(* CODESYS project SZ10-12 PROJ.project

Project tree, tasks and I/O mapping:
  Device : CPX-CEC-S1-V3, Festo AG & Co. KG, order no. 3472425, version 3.5.7.37
      unmapped channels: Rotary switch
    application Application
      libraries: Standard, * (System)
      task MainTask (cyclic, interval t#20ms, priority 20) calls PLC_PRG
      program PLC_PRG [SFC]: Step0_active, Step7_active, Step1_active, Step2_active, Step3_active, Step4_active, Step6_active, Step5_active, Step8_active, Init_active, Step9_active, Step10_active, Step11_active, Step12_active, Step14_active, Step15_active, Step16_active, Step17_active, Step18_active, Step19_active, Step20_active, Step21_active, Step30_active, Step31_active, Step32_active, Step33_active, Step36_active
      global variables GVL
    PLC_Diagnosis : PLC-Diagnosis, Festo AG & Co. KG, version 3.5.4.1
    CPX_System : CPX_System, Festo AG & Co. KG, order no. 3472425, version 1.258
      CEC_S1_V3 : CEC-S1-V3, Festo AG & Co. KG, order no. 3472425, version 1.258
          settings:  = 0;  = 169055699865088;  = 1107404992;  = 16777215;  = 16885952;  = 13959210;  = 1f58c199;  = 5
      _8DI_8DO : 8DI/8DO, Festo AG & Co. KG, order no. 526257, version 1.258
          settings:  = 0;  = 1;  = 1;  = 1;  = 1;  = 0;  = 1;  = 1;  = 0;  = 0;  = 0;  = 0;  = 0;  = 0;  = 0;  = 0;  = 0;  = 0;  = 0;  = 0;  = 0;  = 0;  = 0;  = 0;  = 0;  = 0;  = 0;  = 0;  = 0;  = 0;  = 0;  = 0;  = 0;  = 0;  = 0;  = 0;  = 0;  = 0;  = 0;  = 0;
             = 0;  = 0;  = 0;  = 0;  = 0;  = 0;  = 0;  = 0;  = 0;  = 0;  = 0;  = 0;  = 0;  = 0;  = 0;  = 0;  = 0;  = 0;  = 0;  = 0;  = 0;  = 0;  = 0;  = 0;  = 0;  = 0;  = 0;  = 0;  = 0;  = 0;  = 0;  = 0;  = 0;  = 0;  = 0;  = 0;  = 0;  = 0;  = 0;  = 0;
             = 576751027668385792;  = 'PI%i.0.0.1=1';  = 'PI%i.0.1.1=1';  = 'PI%i.0.2.1=1';  = 'PI%i.1.0.1=1';  = 'PI%i.1.1.1=0';  = 'PI%i.1.4.2=1';  = 'PI%i.1.6.2=1';  = 'PI%i.6.0.1=0';  = 'PI%i.6.1.1=0';  = 'PI%i.6.2.1=0';  = 'PI%i.6.3.1=0';  = 'PI%i.6.4.1=0';  = 'PI%i.6.5.1=0';  = 'PI%i.6.6.1=0';  = 'PI%i.6.7.1=0';  = dd3e3128;  = 6
          unmapped channels: Input 0, Output 0
      _8DI_8DO_1 : 8DI/8DO, Festo AG & Co. KG, order no. 526257, version 1.258
          settings:  = 0;  = 1;  = 1;  = 1;  = 1;  = 0;  = 1;  = 1;  = 0;  = 0;  = 0;  = 0;  = 0;  = 0;  = 0;  = 0;  = 0;  = 0;  = 0;  = 0;  = 0;  = 0;  = 0;  = 0;  = 0;  = 0;  = 0;  = 0;  = 0;  = 0;  = 0;  = 0;  = 0;  = 0;  = 0;  = 0;  = 0;  = 0;  = 0;  = 0;
             = 0;  = 0;  = 0;  = 0;  = 0;  = 0;  = 0;  = 0;  = 0;  = 0;  = 0;  = 0;  = 0;  = 0;  = 0;  = 0;  = 0;  = 0;  = 0;  = 0;  = 0;  = 0;  = 0;  = 0;  = 0;  = 0;  = 0;  = 0;  = 0;  = 0;  = 0;  = 0;  = 0;  = 0;  = 0;  = 0;  = 0;  = 0;  = 0;  = 0;
             = 576751027668385792;  = 'PI%i.0.0.1=1';  = 'PI%i.0.1.1=1';  = 'PI%i.0.2.1=1';  = 'PI%i.1.0.1=1';  = 'PI%i.1.1.1=0';  = 'PI%i.1.4.2=1';  = 'PI%i.1.6.2=1';  = 'PI%i.6.0.1=0';  = 'PI%i.6.1.1=0';  = 'PI%i.6.2.1=0';  = 'PI%i.6.3.1=0';  = 'PI%i.6.4.1=0';  = 'PI%i.6.5.1=0';  = 'PI%i.6.6.1=0';  = 'PI%i.6.7.1=0';  = dd3e312f;  = 6
          unmapped channels: Input 0, Output 0
      _2AI : 2AI, Festo AG & Co. KG, order no. 526168, version 1.258
          settings:  = 0;  = 1;  = 1;  = 1;  = 1;  = 128;  = 128;  = 0;  = 0;  = 0;  = 0;  = 0;  = 0;  = 4095;  = 4095;  = 0;  = 0;  = 0;  = 0;  = 148618787711614976;  = 'PI%i.0.0.1=1';  = 'PI%i.0.7.1=1';  = 'PI%i.1.0.1=1';  = 'PI%i.3.0.2=1';  = 'PI%i.6.0.8=128';  = 'PI%i.7.0.8=128';  = 'PI%i.8.0.4=0';  = 'PI%i.8.4.4=0';  = 'PI%i.9.0.4=0';  = 'PI%i.9.4.4=0';  = 'PI%i.10.0.16=0';  = 'PI%i.12.0.16=0';  = 'PI%i.14.0.16=4095';  = 'PI%i.16.0.16=4095';  = dd3e2ea6;  = 15
          unmapped channels: Input 0, Input 1
      _2AO : 2AO, Festo AG & Co. KG, order no. 526170, version 1.258
          settings:  = 0;  = 1;  = 1;  = 1;  = 0;  = 1;  = 135;  = 135;  = 0;  = 0;  = 0;  = 0;  = 4095;  = 4095;  = 0;  = 0;  = 0;  = 0;  = 0;  = 0;  = 0;  = 0;  = 0;  = 0;  = 0;  = 0;  = 2267751186432;  = 'PI%i.0.1.1=1';  = 'PI%i.0.7.1=1';  = 'PI%i.1.1.1=1';  = 'PI%i.1.3.1=0';  = 'PI%i.3.4.2=1';  = 'PI%i.6.0.8=135';  = 'PI%i.7.0.8=135';  = 'PI%i.8.0.4=0';  = 'PI%i.8.4.4=0';  = 'PI%i.9.0.16=0';  = 'PI%i.11.0.16=0';  = 'PI%i.13.0.16=4095';  = 'PI%i.15.0.16=4095';
             = dd3e3a6a;  = 18
          unmapped channels: Output 0, Output 1
      MPA1S : MPA1S, Festo AG & Co. KG, order no. 533360, version 1.258
          settings:  = 0;  = 1;  = 0;  = 0;  = 0;  = 0;  = 0;  = 0;  = 0;  = 0;  = 0;  = 0;  = 0;  = 0;  = 0;  = 0;  = 0;  = 0;  = 0;  = 0;  = 0;  = 0;  = 0;  = 0;  = 0;  = 0;  = 0;  = 0;  = 0;  = 0;  = 0;  = 0;  = 0;  = 0;  = 0;  = 0;  = 0;  = 0;  = 0;  = 0;
             = 0;  = 0;  = 0;  = 0;  = 0;  = 0;  = 0;  = 0;  = 0;  = 0;  = 8800393363456;  = 'PI%i.0.2.1=1';  = dd3d905e;  = 9
          unmapped channels: Output 0
*)

// Device/Application/GVL
VAR_GLOBAL
	START AT %IX2.0: BOOL;
	STOP AT %IX2.4: BOOL;
	KETTO AT %IX2.2: BOOL;
	HAROM AT %IX2.6: BOOL;
	NEGY AT %IX2.7: BOOL;
	XBALH AT %IX1.0: BOOL;
	XJOBBH AT %IX1.4: BOOL;
	YBENT AT %IX1.5: BOOL;
	YKINT AT %IX1.1: BOOL;
	ZLENT AT %IX1.2: BOOL;
	ZFENT AT %IX1.6: BOOL;
	MEGFZ AT %IX1.7: BOOL;
	MEGFNY AT %IX1.3: BOOL;
	XBALRA AT %QX0.4: BOOL;
	XJOBBRA AT %QX0.0: BOOL;
	YBE AT %QX0.5: BOOL;
	YKI AT %QX0.1: BOOL;
	ZLE AT %QX0.6: BOOL;
	ZFEL AT %QX0.2: BOOL;
	FORG AT %QX0.7: BOOL;
	MEGF AT %QX0.3: BOOL;
	FURAT AT %IX2.1: BOOL;
	FURAT1: BOOL;
	FURAT2: BOOL;
	KAPCS AT %IX2.5: BOOL;
	FEM: BOOL;
	IND AT %IX2.3: BOOL;
	ZOLD AT %QX1.4: BOOL;
END_VAR

// Device/Application/PLC_PRG
PROGRAM PLC_PRG
VAR
END_VAR

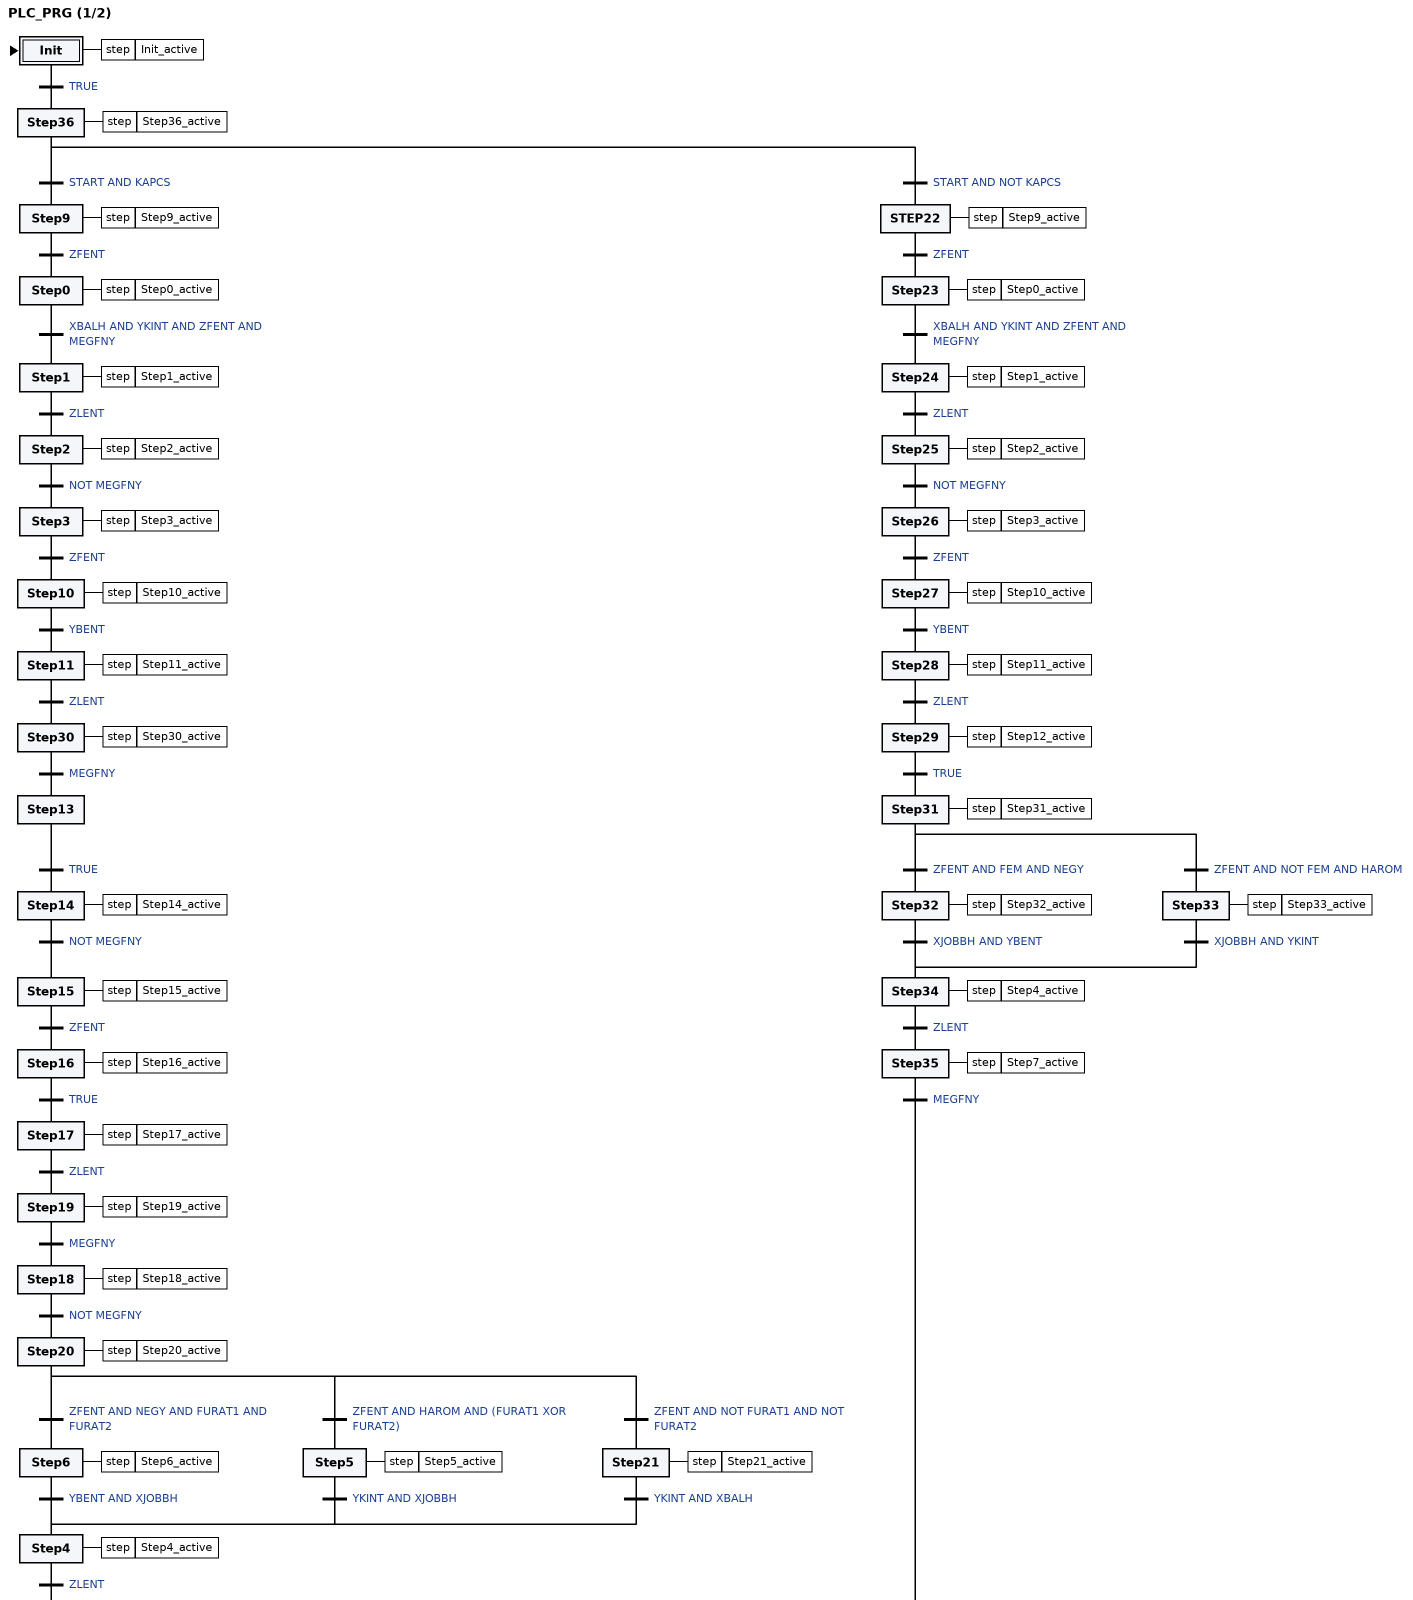
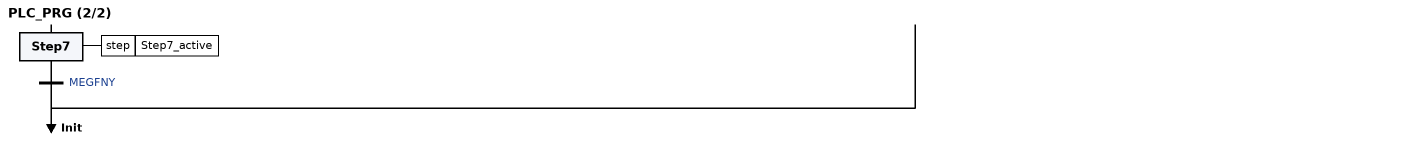
INITIAL_STEP Init:
    Init_active(N);  // step action
END_STEP
TRANSITION FROM Init TO Step36
    := TRUE;
END_TRANSITION
STEP Step36:
    Step36_active(N);  // step action
END_STEP
TRANSITION FROM Step36 TO Step9
    := START AND KAPCS;
END_TRANSITION
STEP Step9:
    Step9_active(N);  // step action
END_STEP
TRANSITION FROM Step9 TO Step0
    := ZFENT;
END_TRANSITION
STEP Step0:
    Step0_active(N);  // step action
END_STEP
TRANSITION FROM Step0 TO Step1
    := XBALH AND YKINT AND ZFENT AND MEGFNY;
END_TRANSITION
STEP Step1:
    Step1_active(N);  // step action
END_STEP
TRANSITION FROM Step1 TO Step2
    := ZLENT;
END_TRANSITION
STEP Step2:
    Step2_active(N);  // step action
END_STEP
TRANSITION FROM Step2 TO Step3
    := NOT MEGFNY;
END_TRANSITION
STEP Step3:
    Step3_active(N);  // step action
END_STEP
TRANSITION FROM Step3 TO Step10
    := ZFENT;
END_TRANSITION
STEP Step10:
    Step10_active(N);  // step action
END_STEP
TRANSITION FROM Step10 TO Step11
    := YBENT;
END_TRANSITION
STEP Step11:
    Step11_active(N);  // step action
END_STEP
TRANSITION FROM Step11 TO Step30
    := ZLENT;
END_TRANSITION
STEP Step30:
    Step30_active(N);  // step action
END_STEP
TRANSITION FROM Step30 TO Step13
    := MEGFNY;
END_TRANSITION
STEP Step13:  // min time T#2S
END_STEP
TRANSITION FROM Step13 TO Step14
    := TRUE;
END_TRANSITION
STEP Step14:
    Step14_active(N);  // step action
END_STEP
TRANSITION FROM Step14 TO Step15
    := NOT MEGFNY;
END_TRANSITION
STEP Step15:
    Step15_active(N);  // step action
END_STEP
TRANSITION FROM Step15 TO Step16
    := ZFENT;
END_TRANSITION
STEP Step16:
    Step16_active(N);  // step action
END_STEP
TRANSITION FROM Step16 TO Step17
    := TRUE;
END_TRANSITION
STEP Step17:
    Step17_active(N);  // step action
END_STEP
TRANSITION FROM Step17 TO Step19
    := ZLENT;
END_TRANSITION
STEP Step19:  // min time T#2s
    Step19_active(N);  // step action
END_STEP
TRANSITION FROM Step19 TO Step18
    := MEGFNY;
END_TRANSITION
STEP Step18:
    Step18_active(N);  // step action
END_STEP
TRANSITION FROM Step18 TO Step20
    := NOT MEGFNY;
END_TRANSITION
STEP Step20:
    Step20_active(N);  // step action
END_STEP
TRANSITION FROM Step20 TO Step6
    := ZFENT AND NEGY AND FURAT1 AND FURAT2;
END_TRANSITION
STEP Step6:
    Step6_active(N);  // step action
END_STEP
TRANSITION FROM Step6 TO Step4
    := YBENT AND XJOBBH;
END_TRANSITION
TRANSITION FROM Step20 TO Step5
    := ZFENT AND HAROM AND (FURAT1 XOR FURAT2);
END_TRANSITION
STEP Step5:
    Step5_active(N);  // step action
END_STEP
TRANSITION FROM Step5 TO Step4
    := YKINT AND XJOBBH;
END_TRANSITION
TRANSITION FROM Step20 TO Step21
    := ZFENT AND NOT FURAT1 AND NOT FURAT2;
END_TRANSITION
STEP Step21:
    Step21_active(N);  // step action
END_STEP
TRANSITION FROM Step21 TO Step4
    := YKINT AND XBALH;
END_TRANSITION
STEP Step4:
    Step4_active(N);  // step action
END_STEP
TRANSITION FROM Step4 TO Step7
    := ZLENT;
END_TRANSITION
STEP Step7:
    Step7_active(N);  // step action
END_STEP
TRANSITION FROM Step7 TO Init
    := MEGFNY;
END_TRANSITION
TRANSITION FROM Step36 TO STEP22
    := START AND NOT KAPCS;
END_TRANSITION
STEP STEP22:
    Step9_active(N);  // step action
END_STEP
TRANSITION FROM STEP22 TO Step23
    := ZFENT;
END_TRANSITION
STEP Step23:
    Step0_active(N);  // step action
END_STEP
TRANSITION FROM Step23 TO Step24
    := XBALH AND YKINT AND ZFENT AND MEGFNY;
END_TRANSITION
STEP Step24:
    Step1_active(N);  // step action
END_STEP
TRANSITION FROM Step24 TO Step25
    := ZLENT;
END_TRANSITION
STEP Step25:
    Step2_active(N);  // step action
END_STEP
TRANSITION FROM Step25 TO Step26
    := NOT MEGFNY;
END_TRANSITION
STEP Step26:
    Step3_active(N);  // step action
END_STEP
TRANSITION FROM Step26 TO Step27
    := ZFENT;
END_TRANSITION
STEP Step27:
    Step10_active(N);  // step action
END_STEP
TRANSITION FROM Step27 TO Step28
    := YBENT;
END_TRANSITION
STEP Step28:
    Step11_active(N);  // step action
END_STEP
TRANSITION FROM Step28 TO Step29
    := ZLENT;
END_TRANSITION
STEP Step29:  // min time T#1s
    Step12_active(N);  // step action
END_STEP
TRANSITION FROM Step29 TO Step31
    := TRUE;
END_TRANSITION
STEP Step31:
    Step31_active(N);  // step action
END_STEP
TRANSITION FROM Step31 TO Step32
    := ZFENT AND FEM AND NEGY;
END_TRANSITION
STEP Step32:
    Step32_active(N);  // step action
END_STEP
TRANSITION FROM Step32 TO Step34
    := XJOBBH AND YBENT;
END_TRANSITION
TRANSITION FROM Step31 TO Step33
    := ZFENT AND NOT FEM AND HAROM;
END_TRANSITION
STEP Step33:
    Step33_active(N);  // step action
END_STEP
TRANSITION FROM Step33 TO Step34
    := XJOBBH AND YKINT;
END_TRANSITION
STEP Step34:
    Step4_active(N);  // step action
END_STEP
TRANSITION FROM Step34 TO Step35
    := ZLENT;
END_TRANSITION
STEP Step35:
    Step7_active(N);  // step action
END_STEP
TRANSITION FROM Step35 TO Init
    := MEGFNY;
END_TRANSITION

ACTION Step0_active:
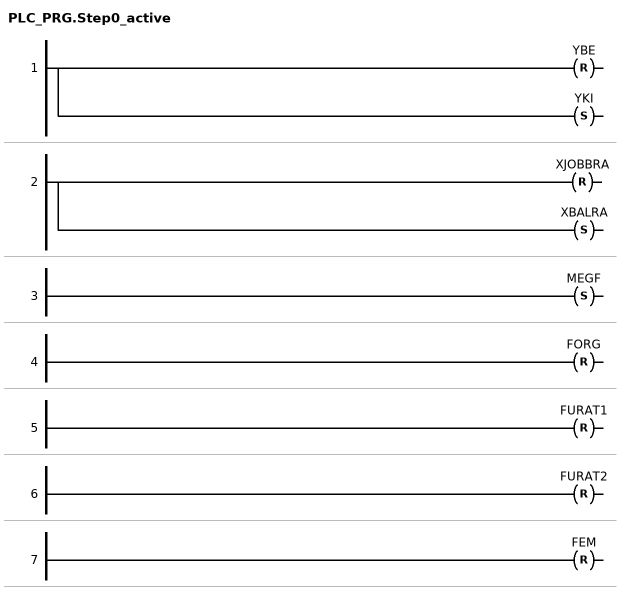
// NETWORK 1
YBE R= TRUE;
YKI S= TRUE;

// NETWORK 2
XJOBBRA R= TRUE;
XBALRA S= TRUE;

// NETWORK 3
MEGF S= TRUE;

// NETWORK 4
FORG R= TRUE;

// NETWORK 5
FURAT1 R= TRUE;

// NETWORK 6
FURAT2 R= TRUE;

// NETWORK 7
FEM R= TRUE;
END_ACTION

ACTION Step7_active:
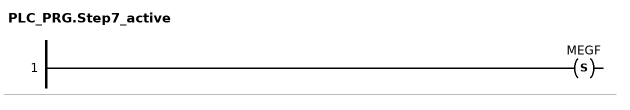
// NETWORK 1
MEGF S= TRUE;
END_ACTION

ACTION Step1_active:
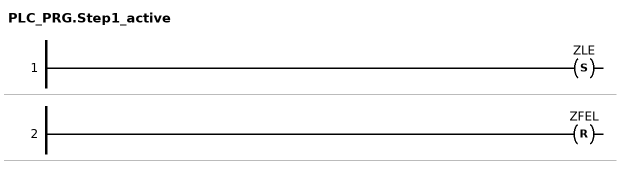
// NETWORK 1
ZLE S= TRUE;

// NETWORK 2
ZFEL R= TRUE;
END_ACTION

ACTION Step2_active:
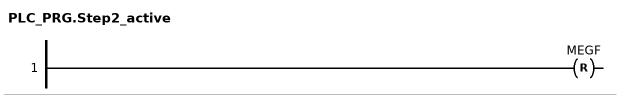
// NETWORK 1
MEGF R= TRUE;
END_ACTION

ACTION Step3_active:
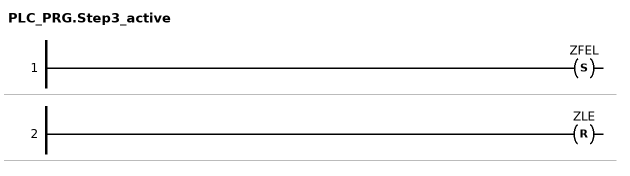
// NETWORK 1
ZFEL S= TRUE;

// NETWORK 2
ZLE R= TRUE;
END_ACTION

ACTION Step4_active:
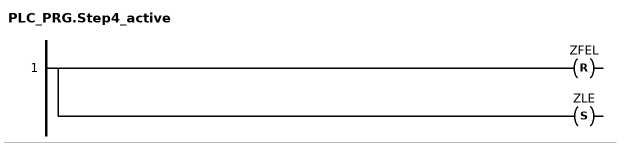
// NETWORK 1
ZFEL R= TRUE;
ZLE S= TRUE;
END_ACTION

ACTION Step6_active:
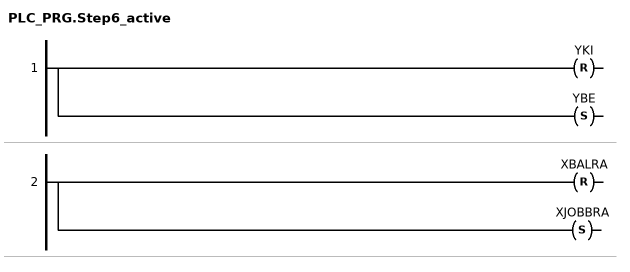
// NETWORK 1
YKI R= TRUE;
YBE S= TRUE;

// NETWORK 2
XBALRA R= TRUE;
XJOBBRA S= TRUE;
END_ACTION

ACTION Step5_active:
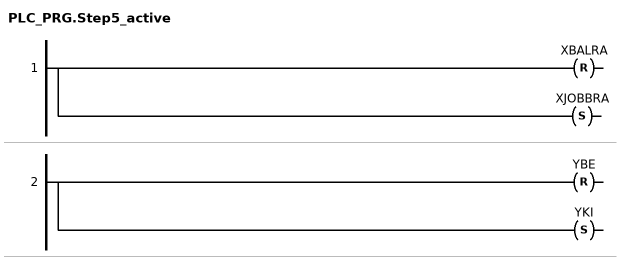
// NETWORK 1
XBALRA R= TRUE;
XJOBBRA S= TRUE;

// NETWORK 2
YBE R= TRUE;
YKI S= TRUE;
END_ACTION

ACTION Step8_active:
// NETWORK 1
END_ACTION

ACTION Init_active:

END_ACTION

ACTION Step9_active:
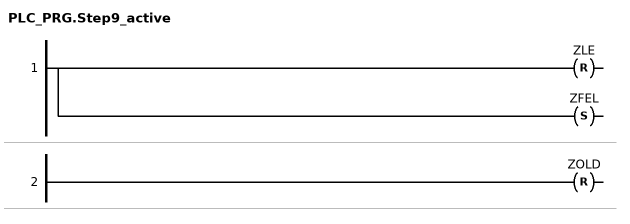
// NETWORK 1
ZLE R= TRUE;
ZFEL S= TRUE;

// NETWORK 2
ZOLD R= TRUE;
END_ACTION

ACTION Step10_active:
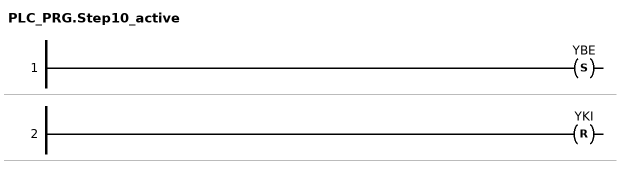
// NETWORK 1
YBE S= TRUE;

// NETWORK 2
YKI R= TRUE;
END_ACTION

ACTION Step11_active:
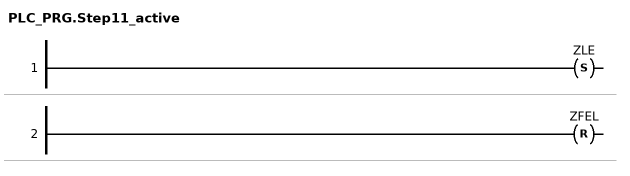
// NETWORK 1
ZLE S= TRUE;

// NETWORK 2
ZFEL R= TRUE;
END_ACTION

ACTION Step12_active:
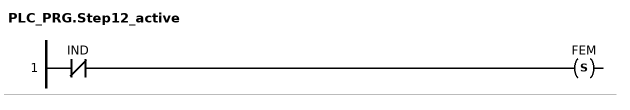
// NETWORK 1
FEM S= NOT IND;
END_ACTION

ACTION Step14_active:
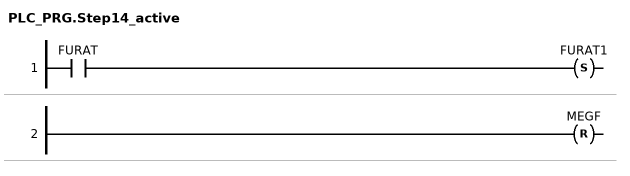
// NETWORK 1
FURAT1 S= FURAT;

// NETWORK 2
MEGF R= TRUE;
END_ACTION

ACTION Step15_active:
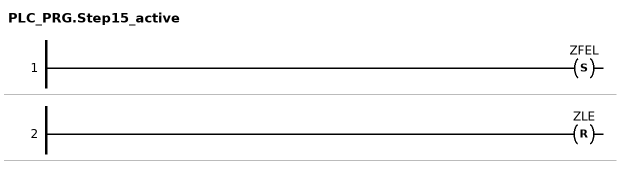
// NETWORK 1
ZFEL S= TRUE;

// NETWORK 2
ZLE R= TRUE;
END_ACTION

ACTION Step16_active:
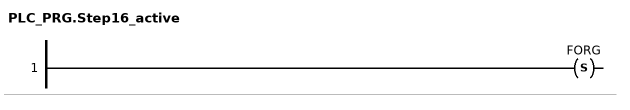
// NETWORK 1
FORG S= TRUE;
END_ACTION

ACTION Step17_active:
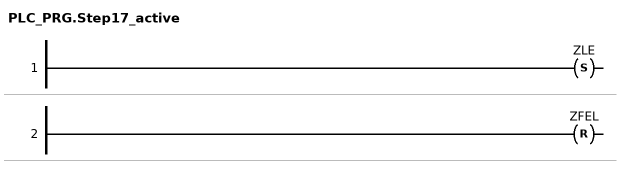
// NETWORK 1
ZLE S= TRUE;

// NETWORK 2
ZFEL R= TRUE;
END_ACTION

ACTION Step18_active:
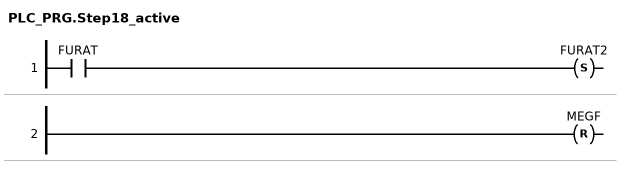
// NETWORK 1
FURAT2 S= FURAT;

// NETWORK 2
MEGF R= TRUE;
END_ACTION

ACTION Step19_active:
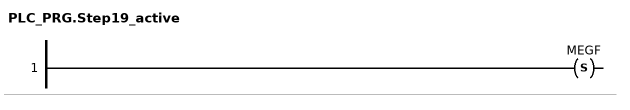
// NETWORK 1
MEGF S= TRUE;
END_ACTION

ACTION Step20_active:
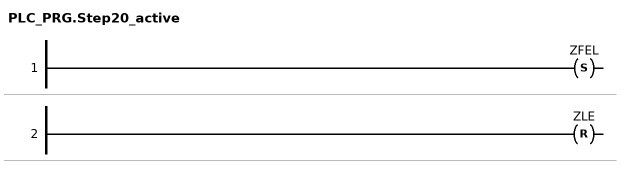
// NETWORK 1
ZFEL S= TRUE;

// NETWORK 2
ZLE R= TRUE;
END_ACTION

ACTION Step21_active:
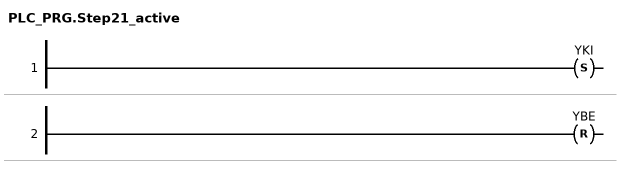
// NETWORK 1
YKI S= TRUE;

// NETWORK 2
YBE R= TRUE;
END_ACTION

ACTION Step30_active:
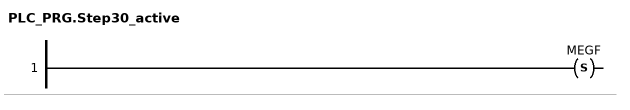
// NETWORK 1
MEGF S= TRUE;
END_ACTION

ACTION Step31_active:
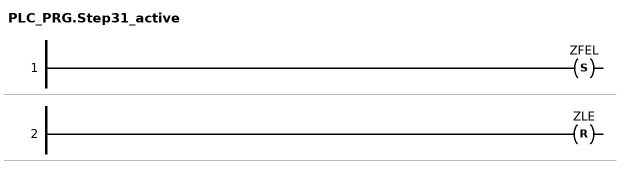
// NETWORK 1
ZFEL S= TRUE;

// NETWORK 2
ZLE R= TRUE;
END_ACTION

ACTION Step32_active:
